(*
SPDX-FileCopyrightText: © 2026 Oleksandr Tiutyk <trofimich@gmail.com>
SPDX-License-Identifier: MIT
License: https://opensource.org/license/mit
*)

{attribute 'no_explicit_call' := 'do not call this function block directly'} 
PROGRAM LongTimes
VAR CONSTANT
	MIN_VALUE : LTIME := LTIME#0S;
	MAX_VALUE : LTIME := LTIME#213503D23H34M33S709MS551US615NS;
END_VAR
VAR
	{attribute 'hide'} 
	_ClassName : STRING := __POUNAME();
END_VAR

{attribute 'monitoring' := 'call'}
PROPERTY ClassName : REFERENCE TO STRING
GET
ClassName REF= _ClassName;
END_GET
END_PROPERTY

METHOD FromDays : LTIME
VAR_INPUT
	timeInDays : LREAL;
END_VAR
FromDays := TO_LTIME(timeInDays * 86_400_000_000_000);
END_METHOD

METHOD FromHours : LTIME
VAR_INPUT
	timeInHours : LREAL;
END_VAR
FromHours := TO_LTIME(timeInHours * 3_600_000_000_000);
END_METHOD

METHOD FromMicroseconds : LTIME
VAR_INPUT
	timeInMicroseconds : LREAL;
END_VAR
FromMicroseconds := TO_LTIME(timeInMicroseconds * 1_000);
END_METHOD

METHOD FromMiliseconds : LTIME
VAR_INPUT
	timeInMiliseconds : LREAL;
END_VAR
FromMiliseconds := TO_LTIME(timeInMiliseconds * 1_000_000);
END_METHOD

METHOD FromMinutes : LTIME
VAR_INPUT
	timeInMinutes : LREAL;
END_VAR
FromMinutes := TO_LTIME(timeInMinutes * 60_000_000_000);
END_METHOD

METHOD FromNanoseconds : LTIME
VAR_INPUT
	timeInNanoseconds : LREAL;
END_VAR
FromNanoseconds := TO_LTIME(timeInNanoseconds);
END_METHOD

METHOD FromSeconds : LTIME
VAR_INPUT
	timeInSeconds : LREAL;
END_VAR
FromSeconds := TO_LTIME(timeInSeconds * 1_000_000_000);
END_METHOD

{attribute 'monitoring' := 'call'}
PROPERTY NamespaceName : REFERENCE TO STRING
GET
NamespaceName REF= CurrentNamespace.Name;
END_GET
END_PROPERTY

END_PROGRAM

(* stored: Version 1.1.0.1
   POU LongTimes: Id {263e7e24-5aea-46bd-812b-7ae09f701d7e}, SpecialFunc None
   Property ClassName: Id {f8be15f5-076c-48ca-bf4d-3a9e95f8c7a2}
   Get Get: Id {0117bffd-f478-4b70-b5bc-46a0d24d6d47}
   Method FromDays: Id {378c3778-10dd-431b-be55-69536192d36c}
   Method FromHours: Id {6d48b5e3-f6f9-4cda-bd2f-7268aac24b56}
   Method FromMicroseconds: Id {9de3e4e6-2a06-42e2-ab0e-f0722937ecc1}
   Method FromMiliseconds: Id {60adc2ea-a38d-47d4-a474-7a2d67c4313f}
   Method FromMinutes: Id {4864dc88-5558-4377-87d4-5c0d0b7e14a0}
   Method FromNanoseconds: Id {9b282456-af17-4b2c-b3b4-1526186f44af}
   Method FromSeconds: Id {aaba609a-b89b-4cb6-ad92-158daadb2ebe}
   Property NamespaceName: Id {6cc57616-a14c-441b-bc54-f3c5ba4249d0}
   Get Get: Id {66442e2b-6586-4c7d-b0cf-573d7538d031} *)
